{attribute 'qualified_only'}
{attribute 'strict'}
TYPE E_TestEnum :
(
	Disabled 	:= 0,
	Starting 	:= 50,
	Running 	:= 100,
	Stopping	:= 200	
);
END_TYPE

(* stored: Version 1.1.0.1, ProductVersion 3.1.4024.12
   DUT E_TestEnum: Id {9ff8884d-dce7-404c-9edb-d78d08cd7196} *)
